(* PLC project plc, Dassault Systèmes ControlBuild 2024x Refresh1 *)
(* stored: creationDateTime 2024-04-09T14:41:20-01:00 *)

PROGRAM flask_motion_app.plc

(* FBD diagram, written out as Structured Text *)
END_PROGRAM
